(* CODESYS project Domains.library
   Company: _
   DefaultNamespace: Domains
   Title: Domains
   Placeholder: _Domains
   Author: Krystian Lis et al.
   Description: Each Domain should have a number of standard browsable components.
   Version: 1.0.0

Project tree, tasks and I/O mapping:
  libraries: Broadcast, * (_); Debug, * (_); Flags, * (_); States, * (_); Tags, * (_); Tc2_Standard, * (Beckhoff Automation GmbH); Tc3_Module, * (Beckhoff Automation GmbH); Results, * (_)
  Domain/
    Iter/
      function block DomainIter [ST]: FB_init, First, Get, GetPos, Last, Next, Peek, PeekBack, PeekPos, Prev
      interface I_DomainIter: First, Get, GetPos, Last, Next, Peek, PeekBack, PeekPos, Prev
    global variables _Domain
    function block Domain [ST]: Attach, FB_init, Next, Prev, state, ToDebug, Flags, Recs, Signals, Smgr, Tag
    interface I_Domain: Flags, Recs, Signals, Smgr
    interface I_DomainNode: Attach, Next, Prev, state
*)

// Domain/_Domain
{attribute 'qualified_only'}
VAR_GLOBAL INTERNAL
	iFirst			: I_DomainNode;
	iLast			: I_DomainNode;
END_VAR

// Domain/Iter/DomainIter
FUNCTION_BLOCK DomainIter
VAR
	_iPointer		: I_DomainNode;
	_eState			: Results.Result;
END_VAR

//FB_Init is always available implicitly and it is used primarily for initialization.
//The return value is not evaluated. For a specific influence, you can also declare the
//methods explicitly and provide additional code there with the standard initialization
//code. You can evaluate the return value.
METHOD FB_Init: BOOL
VAR_INPUT
    bInitRetains: BOOL; // TRUE: the retain variables are initialized (reset warm / reset cold)
    bInCopyCode: BOOL;  // TRUE: the instance will be copied to the copy code afterward (online change)   
END_VAR
_iPointer := _Domain.iFirst;
IF _iPointer <> 0 THEN
	_eState := Results.Ok;
ELSE
	_eState := Results.None;
END_IF
END_METHOD

METHOD First : Results.Result
VAR_OUTPUT
	iDomain		: I_Domain;
END_VAR
_iPointer := _Domain.iFirst;
IF _iPointer <> 0 THEN
	_eState := Results.Ok;
ELSE
	_eState := Results.None;
END_IF
First := _eState;
iDomain := _iPointer;
END_METHOD

METHOD Get : Results.Result
VAR_OUTPUT
	iDomain		: I_Domain;
END_VAR
Get := _eState;
iDomain := _iPointer;
END_METHOD

METHOD GetPos : Results.Result
VAR_INPUT
	nPos		: UDINT;
END_VAR
VAR_OUTPUT
	iDomain		: I_Domain;
END_VAR
VAR
	i			: UDINT;
END_VAR
_iPointer := _Domain.iFirst;
IF _iPointer = 0 THEN
    _eState := Results.None;
   	GetPos := _eState;
	RETURN;
END_IF

IF nPos = 0 THEN
	_eState := Results.Ok;
	iDomain := _iPointer;
	GetPos := _eState;
	RETURN;
END_IF

FOR i := 0 TO nPos - 1 DO
    _iPointer := _iPointer.Next;
    IF _iPointer = 0 THEN
		_eState := Results.None;
        GetPos := _eState;
    END_IF
END_FOR

_eState := Results.Ok;
GetPos := _eState;
iDomain := _iPointer;
END_METHOD

METHOD Last : Results.Result
VAR_OUTPUT
	iDomain		: I_Domain;
END_VAR
_iPointer := _Domain.iLast;
IF _iPointer <> 0 THEN
	_eState := Results.Ok;
ELSE
	_eState := Results.None;
END_IF
Last := _eState;
iDomain := _iPointer;
END_METHOD

METHOD Next : Results.Result
VAR_OUTPUT
	iDomain		: I_Domain;
END_VAR
IF _eState <> Results.Ok THEN
	Next := Results.None;
	RETURN;
END_IF

_iPointer := _iPointer.Next;
IF _iPointer <> 0 THEN
	_eState := Results.Ok;
ELSE
	_eState := Results.None;
END_IF
Next := _eState;
iDomain := _iPointer;
END_METHOD

METHOD Peek : Results.Result
VAR_OUTPUT
	iDomain		: I_Domain;
END_VAR
IF _eState <> Results.Ok THEN
	Peek := Results.None;
	RETURN;
END_IF

iDomain := _iPointer.Next;
IF iDomain <> 0 THEN
	_eState := Results.Ok;
ELSE
	_eState := Results.None;
END_IF
Peek := _eState;
END_METHOD

METHOD PeekBack : Results.Result
VAR_OUTPUT
	iDomain		: I_Domain;
END_VAR
IF _eState <> Results.Ok THEN
	PeekBack := Results.None;
	RETURN;
END_IF

iDomain := _iPointer.Prev;
IF iDomain <> 0 THEN
	_eState := Results.Ok;
ELSE
	_eState := Results.None;
END_IF
PeekBack := _eState;
END_METHOD

METHOD PeekPos : Results.Result
VAR_INPUT
	nPos		: UDINT;
END_VAR
VAR_OUTPUT
	iDomain		: I_Domain;
END_VAR
VAR
	i			: UDINT;
	_iNode		: I_DomainNode;
END_VAR
_iNode := _Domain.iFirst;
IF _iNode = 0 THEN
    _eState := Results.None;
   	PeekPos := _eState;
	RETURN;
END_IF

IF nPos = 0 THEN
	_eState := Results.Ok;
	iDomain := _iNode;
	PeekPos := _eState;
	RETURN;
END_IF

FOR i := 0 TO nPos - 1 DO
    _iNode := _iNode.Next;
    IF _iNode = 0 THEN
		_eState := Results.None;
        PeekPos := _eState;
    END_IF
END_FOR

_eState := Results.Ok;
PeekPos := _eState;
iDomain := _iNode;
END_METHOD

METHOD Prev : Results.Result
VAR_OUTPUT
	iDomain		: I_Domain;
END_VAR
IF _eState <> Results.Ok THEN
	Prev := Results.None;
	RETURN;
END_IF

_iPointer := _iPointer.Prev;
IF _iPointer <> 0 THEN
	_eState := Results.Ok;
ELSE
	_eState := Results.None;
END_IF
Prev := _eState;
iDomain := _iPointer;
END_METHOD

END_FUNCTION_BLOCK

// Domain/I_DomainNode
INTERFACE INTERNAL I_DomainNode EXTENDS I_Domain,

METHOD INTERNAL Attach : Results.Result
VAR_INPUT
	iNode		: I_DomainNode;
END_VAR
END_METHOD

PROPERTY INTERNAL Next : I_DomainNode
GET
END_GET
END_PROPERTY

PROPERTY INTERNAL Prev : I_DomainNode
GET
END_GET
END_PROPERTY

PROPERTY INTERNAL state : Results.Result
GET
END_GET
SET
END_SET
END_PROPERTY

END_INTERFACE

// Domain/I_Domain
INTERFACE I_Domain EXTENDS Debug.I_Debug, Tags.I_Tagged

PROPERTY Flags : Flags.I_FlagList
GET
END_GET
END_PROPERTY

PROPERTY Recs : Broadcast.I_ReceiverList
GET
END_GET
END_PROPERTY

PROPERTY Signals : Broadcast.I_SignalList
GET
END_GET
END_PROPERTY

PROPERTY Smgr : States.I_StateManager
GET
END_GET
END_PROPERTY

END_INTERFACE

// Domain/Iter/I_DomainIter
INTERFACE I_DomainIter

METHOD First : Results.Result
VAR_OUTPUT
	iDomain		: I_Domain;
END_VAR
END_METHOD

METHOD Get : Results.Result
VAR_OUTPUT
	iDomain		: I_Domain;
END_VAR
END_METHOD

METHOD GetPos : Results.Result
VAR_INPUT
	nPos		: UDINT;
END_VAR
VAR_OUTPUT
	iDomain		: I_Domain;
END_VAR
END_METHOD

METHOD Last : Results.Result
VAR_OUTPUT
	iDomain		: I_Domain;
END_VAR
END_METHOD

METHOD Next : Results.Result
VAR_OUTPUT
	iDomain		: I_Domain;
END_VAR
END_METHOD

METHOD Peek : Results.Result
VAR_OUTPUT
	iDomain		: I_Domain;
END_VAR
END_METHOD

METHOD PeekBack : Results.Result
VAR_OUTPUT
	iDomain		: I_Domain;
END_VAR
END_METHOD

METHOD PeekPos : Results.Result
VAR_INPUT
	nPos		: UDINT;
END_VAR
VAR_OUTPUT
	iDomain		: I_Domain;
END_VAR
END_METHOD

METHOD Prev : Results.Result
VAR_OUTPUT
	iDomain		: I_Domain;
END_VAR
END_METHOD

END_INTERFACE

// Domain/Domain
FUNCTION_BLOCK FINAL Domain IMPLEMENTS I_DomainNode;
VAR
	_fbTag			: Tags.Tag;
	_iDomain		: I_Domain;
	_iNext			: I_DomainNode;
	_iPrev			: I_DomainNode;
	
	_eState			: Results.Result;
END_VAR

METHOD INTERNAL Attach : Results.Result
VAR_INPUT
	iNode			: I_DomainNode;
END_VAR
VAR
	_iThis			: I_DomainNode := THIS^;
END_VAR


IF iNode = 0 THEN
	Debug.DebugMsg(0, Tc2_Standard.CONCAT(__POUNAME(), ': Itf = 0!'));
	RETURN;
END_IF

IF _iThis <> _Domain.iLast THEN
	Debug.DebugMsg(ToDebug(), Tc2_Standard.CONCAT(__POUNAME(), ': Is not the last node!'));
	RETURN;
END_IF

IF Results.IsSome(iNode.state) THEN
	Debug.DebugMsg(iNode.ToDebug(), Tc2_Standard.CONCAT(__POUNAME(), ': Has already been added!'));
	RETURN;
END_IF

_Domain.iLast := iNode;
_iNext := iNode;
END_METHOD

//FB_Init is always available implicitly and it is used primarily for initialization.
//The return value is not evaluated. For a specific influence, you can also declare the
//methods explicitly and provide additional code there with the standard initialization
//code. You can evaluate the return value.
METHOD FB_Init: BOOL
VAR_INPUT
    bInitRetains: BOOL; // TRUE: the retain variables are initialized (reset warm / reset cold)
    bInCopyCode: BOOL;  // TRUE: the instance will be copied to the copy code afterward (online change)

	iDomain			: I_Domain; 
END_VAR
IF Results.IsSome(_eState) THEN
	RETURN;
END_IF

IF (_iDomain := iDomain) = 0 THEN
	_eState := Results.Err.Itf0;
	Debug.DebugMsg(THIS^, Tc2_Standard.CONCAT(__POUNAME(), ': Itf = 0!'));
	RETURN;
END_IF



IF _Domain.iLast <> 0 THEN
	IF Results.IsErr(_Domain.iLast.Attach(THIS^), eCarry => _eState) THEN
		Debug.DebugMsg(THIS^, Tc2_Standard.CONCAT(__POUNAME(), ': Error Inside!'));
	END_IF
ELSE
	_Domain.iFirst := THIS^;
	_Domain.iLast := THIS^;
	_eState := Results.Ok;
END_IF
END_METHOD

PROPERTY INTERNAL Next : I_DomainNode
GET
Next := _iNext;
END_GET
END_PROPERTY

PROPERTY INTERNAL Prev : I_DomainNode
GET
Prev := _iPrev;
END_GET
END_PROPERTY

PROPERTY INTERNAL state : Results.Result
GET
state := _eState;
END_GET
SET
IF Results.IsNone(_eState) THEN
	_eState := state;
END_IF
END_SET
END_PROPERTY

METHOD ToDebug : Debug.I_Debug
ToDebug := THIS^;
END_METHOD

PROPERTY Flags : Flags.I_FlagList
GET
Flags := _iDomain.Flags;
END_GET
END_PROPERTY

PROPERTY Recs : Broadcast.I_ReceiverList
GET
Recs := _iDomain.Recs;
END_GET
END_PROPERTY

PROPERTY Signals : Broadcast.I_SignalList
GET
Signals := _iDomain.Signals;
END_GET
END_PROPERTY

PROPERTY Smgr : States.I_StateManager
GET
Smgr := _iDomain.Smgr;
END_GET
END_PROPERTY

PROPERTY Tag : Tags.I_Tag
GET
Tag := _iDomain.Tag;
END_GET
END_PROPERTY

END_FUNCTION_BLOCK
